(* IEC 61131-3 sources: AxTestProject/Application, 4 files *)

(* ---- Bulb.st ---- *)
NAMESPACE Application

    CLASS Bulb
        VAR
            m_State : BOOL;
        END_VAR

        METHOD PUBLIC Set
            VAR_INPUT
                value : BOOL;
            END_VAR
            VAR_IN_OUT
                Q : stdLib.SignalHandling.BinOutput;
            END_VAR

            Q.SetQ(value := value);
            m_State := Q.IsOn();
        END_METHOD

        METHOD PUBLIC Toggle
            VAR_IN_OUT
                Q : stdLib.SignalHandling.BinOutput;
            END_VAR
                Q.Toggle();
                m_State := Q.IsOn();
        END_METHOD
    END_CLASS

END_NAMESPACE

(* ---- Motor.st ---- *)
NAMESPACE Application

    CLASS Motor
        VAR
            m_Output : stdLib.SignalHandling.BinOutput;
        END_VAR

        METHOD PUBLIC RefToSetSignal
            VAR_IN_OUT
                Q :  stdLib.SignalHandling.BinOutput;
            END_VAR
            m_Output := Q;

        END_METHOD

        METHOD PUBLIC Start
            m_Output.SetQ(true);
        END_METHOD

        METHOD PUBLIC Stop
            m_Output.SetQ(true);
        END_METHOD

    END_CLASS

END_NAMESPACE

(* ---- PushButton.st ---- *)
NAMESPACE Application

    CLASS PushButton
        VAR
            m_switch : stdLib.SignalHandling.BinSignal;
        END_VAR

        METHOD PUBLIC RefToSetSignal
            VAR_IN_OUT
                switch :  stdLib.SignalHandling.BinSignal;
            END_VAR
            m_switch := switch;

        END_METHOD

        METHOD PUBLIC clicked : BOOL
            VAR_INPUT
            END_VAR
            VAR_TEMP
            END_VAR
            clicked := m_switch.QRis();
                ;
        END_METHOD

        METHOD PUBLIC released : BOOL
            VAR_INPUT
            END_VAR
            VAR_TEMP
            END_VAR
            released := m_switch.QFal();
                ;
        END_METHOD

        METHOD PUBLIC isPressed : BOOL
            VAR_INPUT
            END_VAR
            VAR_TEMP
            END_VAR
            isPressed := m_switch.Q();
                ;
        END_METHOD

        METHOD PUBLIC isRelesed : BOOL
            VAR_INPUT
            END_VAR
            VAR_TEMP
            END_VAR
            isRelesed := NOT(m_switch.Q());
                ;
        END_METHOD

    END_CLASS

END_NAMESPACE

(* ---- TrafficLight.st ---- *)
NAMESPACE Application

    CLASS TrafficLight
        VAR
            m_isInitialized : BOOL;
            m_stateINIT : stdLib.Statemachine.State;
            m_stateRed : stdLib.Statemachine.State;
            m_stateRedYe : stdLib.Statemachine.State;
            m_stateGreen : stdLib.Statemachine.State;
            m_stateYellow : stdLib.Statemachine.State;

            m_lampGreen : Application.Bulb;
            m_lampYellow : Application.Bulb;
            m_lampRed : Application.Bulb;

            m_Signal_0_0_gn : stdLib.SignalHandling.BinOutput;
            m_Signal_0_1_ye : stdLib.SignalHandling.BinOutput;
            m_Signal_0_2_rd : stdLib.SignalHandling.BinOutput;

        END_VAR

        METHOD PUBLIC Execute
            VAR_INPUT
                sysLibTimer : DINT;
            END_VAR
            VAR_OUTPUT
                QRed : BOOL;
                QYellow : BOOL;
                QGreen : BOOL;
            END_VAR

            IF (m_isInitialized) THEN
                m_stateINIT.Execute(sysLibTimer := sysLibTimer);
                m_stateGreen.Execute(sysLibTimer := sysLibTimer);
                m_stateYellow.Execute(sysLibTimer := sysLibTimer);
                m_stateRed.Execute(sysLibTimer := sysLibTimer);
                m_stateRedYe.Execute(sysLibTimer := sysLibTimer);

                this.PhaseInit();
                this.PhaseRed();
                this.PhaseRedYellow();
                this.PhaseGreen();
                this.PhaseYellow();
                this.WriteOutputs(QRed => QRed, QYellow => QYellow, QGreen => QGreen);
            END_IF;

        END_METHOD

        METHOD PhaseInit
            IF (m_stateINIT.IsActive()) THEN
                m_lampGreen.Set(value := TRUE, Q := m_Signal_0_0_gn);
                m_lampYellow.Set(value := TRUE, Q := m_Signal_0_1_ye);
                m_lampRed.Set(value := TRUE, Q := m_Signal_0_2_rd);
            END_IF;
            IF (m_stateINIT.OnTimeout(refNextState := m_stateRed)) THEN
                m_lampGreen.Set(value := FALSE, Q := m_Signal_0_0_gn);
                m_lampYellow.Set(value := FALSE, Q := m_Signal_0_1_ye);
                m_lampRed.Set(value := FALSE, Q := m_Signal_0_2_rd);
            END_IF;
        END_METHOD

        METHOD PhaseRed
            //------------------------------------
            // State Phase --> Red Light
            //------------------------------------
            IF (m_stateRed.OnEntry()) THEN
                m_lampRed.Set(value := true, Q := m_Signal_0_2_rd); // Switch on red light
            END_IF;
            IF (m_stateRed.OnTimeOut(refNextState := m_stateYellow)) THEN
                m_lampRed.Set(value := false, Q := m_Signal_0_2_rd); // Switch off red light
            END_IF;
        END_METHOD

        METHOD PhaseRedYellow
            //------------------------------------
            // State Phase --> Red Yellow
            //------------------------------------

            // implement your code here
            ;
        END_METHOD

        METHOD PhaseGreen

            IF (m_stateGreen.OnEntry()) THEN
                m_lampGreen.Set(value := true, Q := m_Signal_0_0_gn); // Switch on green light
            END_IF;
            IF (m_stateGreen.OnTimeOut(refNextState := m_stateRed)) THEN
                m_lampGreen.Set(value := false, Q := m_Signal_0_0_gn); // Switch off green light
            END_IF;
        END_METHOD

        METHOD PhaseYellow
            IF (m_stateYellow.OnEntry()) THEN
                m_lampYellow.Set(value := true, Q := m_Signal_0_1_ye); // Switch on yellow light
            END_IF;
            IF (m_stateYellow.OnTimeOut(refNextState := m_stateGreen)) THEN
                m_lampYellow.Set(value := false, Q := m_Signal_0_1_ye); // Switch off yellow light
            END_IF;
        END_METHOD

        METHOD WriteOutputs
            VAR_OUTPUT
                QRed : BOOL;
                QYellow : BOOL;
                QGreen : BOOL;
            END_VAR
            m_Signal_0_2_rd.SetQ(QRed);
            m_Signal_0_1_ye.SetQ(QYellow);
            m_Signal_0_0_gn.SetQ(QGreen);
        END_METHOD

        METHOD PUBLIC Initialize
            VAR_INPUT
                durationInitPhase : DINT := DINT#4000; // default 2000ms
                durationRedPhase : DINT := DINT#2000; // default 2000ms
                durationRedYellowPhase : DINT := DINT#2000; // default 2000ms
                durationGreenPhase : DINT := DINT#2000; // default 2000ms
                durationYellowPhase : DINT := DINT#2000; // default 2000ms
            END_VAR

            IF (NOT(m_isInitialized)) THEN
                m_isInitialized := TRUE;

                m_stateINIT.Config(monitoringTime := durationInitPhase);
                m_stateGreen.Config(monitoringTime := durationGreenPhase);
                m_stateYellow.Config(monitoringTime := durationYellowPhase);
                m_stateRedYe.Config(monitoringTime := durationRedYellowPhase);
                m_stateRed.Config(monitoringTime := durationRedPhase);
            END_IF;
        END_METHOD

    END_CLASS
END_NAMESPACE
